ABB RobotStudio station: Lab5_Zhuravlev.rsstn

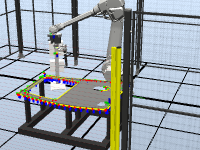
Station GlueStation (saved by RobotStudio 6.8.8307.1040)
Controller IRB4600_20_GlueSystem
  mechanical unit ROB_1: IRB4600_20_250_C_01, 6 joints, base frame (0, 0, 0) mm
Layout (positions relative to the parent item):
  - docking_station [part] at (0, -1345.92, 10) mm, rotated rx 0 ry 0 rz -150 deg
  - SingleDoser [mechanism, from Libraries\SingleDoser.rslib] at (301.98, -1221.72, 1139.56) mm, rotated rx 180 ry -15 rz 15 deg
  - fixture and workpiece [graphiccomponentgroup]
    - door [part]
    - fixture [part]
  - SC_FenceCreator [smart component] at (-1200, -3000, 10) mm
      properties: LengthXside1=4000; LengthXside2=4000; LengthYside1=5300; LengthYside2minus=1500; LengthYside2plus=1500
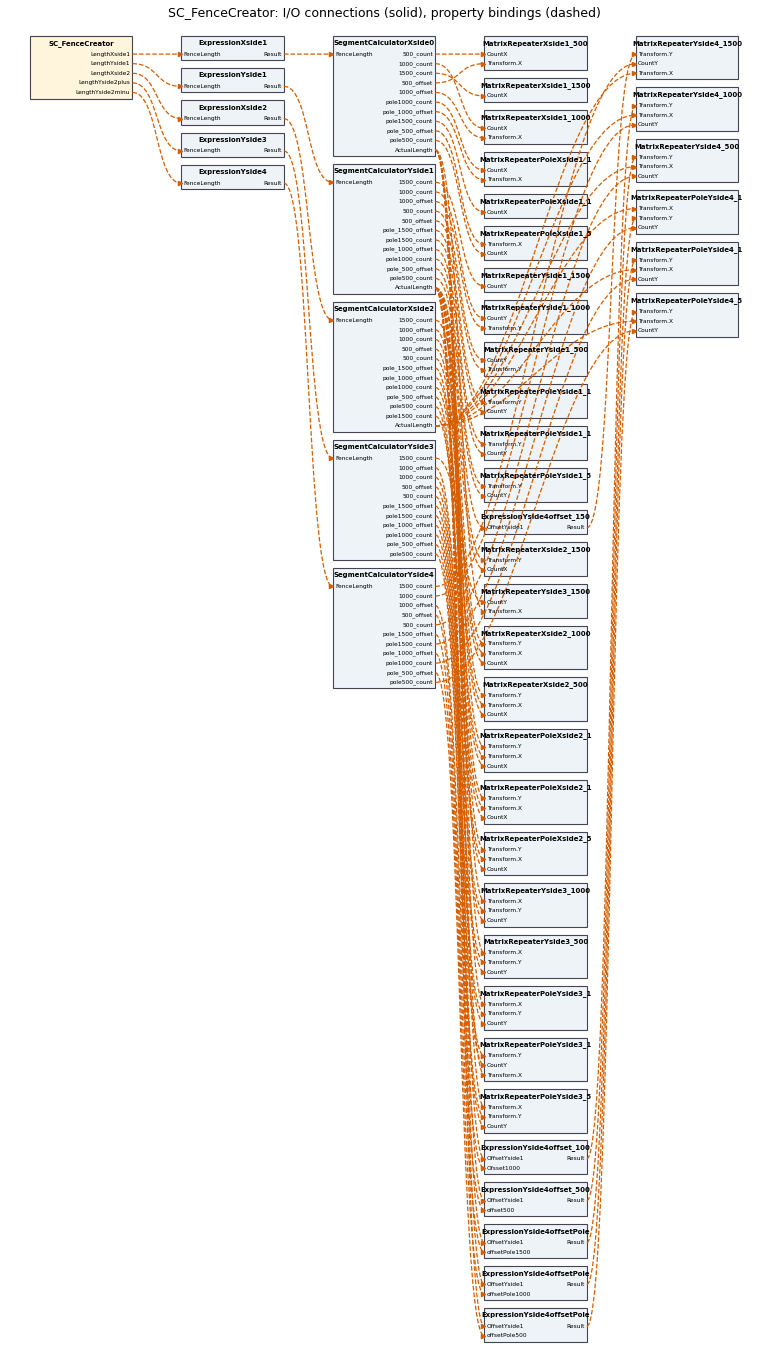
      connections:
        SegmentCalculatorXside0.500_count => MatrixRepeaterXside1_500.CountX
        SegmentCalculatorXside0.1000_count => MatrixRepeaterXside1_1000.CountX
        SegmentCalculatorXside0.1500_count => MatrixRepeaterXside1_1500.CountX
        SegmentCalculatorXside0.500_offset => MatrixRepeaterXside1_500.Transform.X
        SegmentCalculatorXside0.1000_offset => MatrixRepeaterXside1_1000.Transform.X
        SegmentCalculatorXside0.pole1000_count => MatrixRepeaterPoleXside1_1000.CountX
        SegmentCalculatorXside0.pole_1000_offset => MatrixRepeaterPoleXside1_1000.Transform.X
        SegmentCalculatorXside0.pole1500_count => MatrixRepeaterPoleXside1_1500.CountX
        SegmentCalculatorXside0.pole_500_offset => MatrixRepeaterPoleXside1_500.Transform.X
        SegmentCalculatorXside0.pole500_count => MatrixRepeaterPoleXside1_500.CountX
        ExpressionYside1.Result => SegmentCalculatorYside1.FenceLength
        SegmentCalculatorYside1.1500_count => MatrixRepeaterYside1_1500.CountY
        SegmentCalculatorYside1.1000_count => MatrixRepeaterYside1_1000.CountY
        SegmentCalculatorYside1.1000_offset => MatrixRepeaterYside1_1000.Transform.Y
        SegmentCalculatorYside1.500_count => MatrixRepeaterYside1_500.CountY
        SegmentCalculatorYside1.500_offset => MatrixRepeaterYside1_500.Transform.Y
        SegmentCalculatorYside1.pole_1500_offset => MatrixRepeaterPoleYside1_1500.Transform.Y
        SegmentCalculatorYside1.pole1500_count => MatrixRepeaterPoleYside1_1500.CountY
        SegmentCalculatorYside1.pole_1000_offset => MatrixRepeaterPoleYside1_1000.Transform.Y
        SegmentCalculatorYside1.pole1000_count => MatrixRepeaterPoleYside1_1000.CountY
        SegmentCalculatorYside1.pole_500_offset => MatrixRepeaterPoleYside1_500.Transform.Y
        SegmentCalculatorYside1.pole500_count => MatrixRepeaterPoleYside1_500.CountY
        SC_FenceCreator.LengthXside1 => ExpressionXside1.FenceLength
        ExpressionXside2.Result => SegmentCalculatorXside2.FenceLength
        SegmentCalculatorYside1.ActualLength => MatrixRepeaterXside2_1500.Transform.Y
        SegmentCalculatorXside2.1500_count => MatrixRepeaterXside2_1500.CountX
        SegmentCalculatorYside1.ActualLength => MatrixRepeaterXside2_1000.Transform.Y
        SegmentCalculatorXside2.1000_offset => MatrixRepeaterXside2_1000.Transform.X
        SegmentCalculatorXside2.1000_count => MatrixRepeaterXside2_1000.CountX
        SegmentCalculatorYside1.ActualLength => MatrixRepeaterXside2_500.Transform.Y
        SegmentCalculatorXside2.500_offset => MatrixRepeaterXside2_500.Transform.X
        SegmentCalculatorXside2.500_count => MatrixRepeaterXside2_500.CountX
        SegmentCalculatorYside1.ActualLength => MatrixRepeaterPoleXside2_1500.Transform.Y
        SegmentCalculatorXside2.pole_1500_offset => MatrixRepeaterPoleXside2_1500.Transform.X
        SegmentCalculatorYside1.ActualLength => MatrixRepeaterPoleXside2_1000.Transform.Y
        SegmentCalculatorXside2.pole_1000_offset => MatrixRepeaterPoleXside2_1000.Transform.X
        SegmentCalculatorXside2.pole1000_count => MatrixRepeaterPoleXside2_1000.CountX
        SegmentCalculatorYside1.ActualLength => MatrixRepeaterPoleXside2_500.Transform.Y
        SegmentCalculatorXside2.pole_500_offset => MatrixRepeaterPoleXside2_500.Transform.X
        SegmentCalculatorXside2.pole500_count => MatrixRepeaterPoleXside2_500.CountX
        SegmentCalculatorXside2.pole1500_count => MatrixRepeaterPoleXside2_1500.CountX
        SegmentCalculatorYside3.1500_count => MatrixRepeaterYside3_1500.CountY
        ExpressionYside3.Result => SegmentCalculatorYside3.FenceLength
        SegmentCalculatorXside0.ActualLength => MatrixRepeaterYside3_1500.Transform.X
        SegmentCalculatorXside0.ActualLength => MatrixRepeaterYside3_1000.Transform.X
        SegmentCalculatorYside3.1000_offset => MatrixRepeaterYside3_1000.Transform.Y
        SegmentCalculatorYside3.1000_count => MatrixRepeaterYside3_1000.CountY
        SegmentCalculatorXside0.ActualLength => MatrixRepeaterYside3_500.Transform.X
        SegmentCalculatorYside3.500_offset => MatrixRepeaterYside3_500.Transform.Y
        SegmentCalculatorYside3.500_count => MatrixRepeaterYside3_500.CountY
        SegmentCalculatorXside0.ActualLength => MatrixRepeaterPoleYside3_1500.Transform.X
        SegmentCalculatorYside3.pole_1500_offset => MatrixRepeaterPoleYside3_1500.Transform.Y
        SegmentCalculatorYside3.pole1500_count => MatrixRepeaterPoleYside3_1500.CountY
        SegmentCalculatorYside3.pole_1000_offset => MatrixRepeaterPoleYside3_1000.Transform.Y
        SegmentCalculatorYside3.pole1000_count => MatrixRepeaterPoleYside3_1000.CountY
        SegmentCalculatorXside0.ActualLength => MatrixRepeaterPoleYside3_500.Transform.X
        SegmentCalculatorYside3.pole_500_offset => MatrixRepeaterPoleYside3_500.Transform.Y
        SegmentCalculatorYside3.pole500_count => MatrixRepeaterPoleYside3_500.CountY
        SegmentCalculatorXside0.ActualLength => MatrixRepeaterPoleYside3_1000.Transform.X
        ExpressionXside1.Result => SegmentCalculatorXside0.FenceLength
        SC_FenceCreator.LengthYside1 => ExpressionYside1.FenceLength
        SC_FenceCreator.LengthXside2 => ExpressionXside2.FenceLength
        SC_FenceCreator.LengthYside2plus => ExpressionYside3.FenceLength
        SC_FenceCreator.LengthYside2minus => ExpressionYside4.FenceLength
        ExpressionYside4.Result => SegmentCalculatorYside4.FenceLength
        SegmentCalculatorYside1.ActualLength => ExpressionYside4offset_1500.OffsetYside1
        ExpressionYside4offset_1500.Result => MatrixRepeaterYside4_1500.Transform.Y
        SegmentCalculatorYside4.1500_count => MatrixRepeaterYside4_1500.CountY
        SegmentCalculatorXside2.ActualLength => MatrixRepeaterYside4_1500.Transform.X
        SegmentCalculatorYside1.ActualLength => ExpressionYside4offset_1000.OffsetYside1
        ExpressionYside4offset_1000.Result => MatrixRepeaterYside4_1000.Transform.Y
        SegmentCalculatorXside2.ActualLength => MatrixRepeaterYside4_1000.Transform.X
        SegmentCalculatorYside4.1000_count => MatrixRepeaterYside4_1000.CountY
        SegmentCalculatorYside4.1000_offset => ExpressionYside4offset_1000.Ofsset1000
        SegmentCalculatorYside1.ActualLength => ExpressionYside4offset_500.OffsetYside1
        SegmentCalculatorYside4.500_offset => ExpressionYside4offset_500.offset500
        ExpressionYside4offset_500.Result => MatrixRepeaterYside4_500.Transform.Y
        SegmentCalculatorXside2.ActualLength => MatrixRepeaterYside4_500.Transform.X
        SegmentCalculatorYside4.500_count => MatrixRepeaterYside4_500.CountY
        SegmentCalculatorXside2.ActualLength => MatrixRepeaterPoleYside4_1500.Transform.X
        SegmentCalculatorYside1.ActualLength => ExpressionYside4offsetPole_1500.OffsetYside1
        SegmentCalculatorYside4.pole_1500_offset => ExpressionYside4offsetPole_1500.offsetPole1500
        ExpressionYside4offsetPole_1500.Result => MatrixRepeaterPoleYside4_1500.Transform.Y
        SegmentCalculatorYside4.pole1500_count => MatrixRepeaterPoleYside4_1500.CountY
        SegmentCalculatorYside1.ActualLength => ExpressionYside4offsetPole_1000.OffsetYside1
        SegmentCalculatorYside4.pole_1000_offset => ExpressionYside4offsetPole_1000.offsetPole1000
        ExpressionYside4offsetPole_1000.Result => MatrixRepeaterPoleYside4_1000.Transform.Y
        SegmentCalculatorXside2.ActualLength => MatrixRepeaterPoleYside4_1000.Transform.X
        SegmentCalculatorYside4.pole1000_count => MatrixRepeaterPoleYside4_1000.CountY
        SegmentCalculatorYside1.ActualLength => ExpressionYside4offsetPole_500.OffsetYside1
        SegmentCalculatorYside4.pole_500_offset => ExpressionYside4offsetPole_500.offsetPole500
        ExpressionYside4offsetPole_500.Result => MatrixRepeaterPoleYside4_500.Transform.Y
        SegmentCalculatorXside2.ActualLength => MatrixRepeaterPoleYside4_500.Transform.X
        SegmentCalculatorYside4.pole500_count => MatrixRepeaterPoleYside4_500.CountY
    - ExpressionXside1 [smart component, from Libraries\Expression.rslib]
        properties: Expression=FenceLength/1000; FenceLength=4000; Result=4
    - MatrixRepeaterXside1_1500 [smart component, from Libraries\MatrixRepeater.rslib]
        properties: CountX=2; CountY=1; CountZ=1; OffsetX=1.5; OffsetY=0; OffsetZ=0; Source=Panel 2000x1500 X
      - Panel 2000x1500 X [part]
      - Panel 2000x1500 X [part] at (1500, 0, 0) mm
    - MatrixRepeaterXside1_1000 [smart component, from Libraries\MatrixRepeater.rslib] at (3000, 0, 0) mm
        properties: CountX=1; CountY=1; CountZ=1; OffsetX=1; OffsetY=0; OffsetZ=0; Source=Panel 2000x1000 X
      - Panel 2000x1000 X [part]
    - MatrixRepeaterXside1_500 [smart component, from Libraries\MatrixRepeater.rslib] at (4000, 0, 0) mm
        properties: CountX=0; CountY=1; CountZ=1; OffsetX=0.5; OffsetY=0; OffsetZ=0; Source=Panel 2000x500 X
    - MatrixRepeaterPoleXside1_1000 [smart component, from Libraries\MatrixRepeater.rslib] at (4000, 0, 0) mm
        properties: CountX=1; CountY=1; CountZ=1; OffsetX=1; OffsetY=0; OffsetZ=0; Source=Pole
      - Pole [part]
    - Pole [part] at (0, 0, 0) mm
    - SegmentCalculatorXside0 [smart component]
        properties: 1000_count=1; 1000_offset=3; 1500_count=2; 500_count=0; 500_offset=4; ActualLength=4; FenceLength=4; pole_1000_offset=4; pole_1500_offset=0; pole_500_offset=4.5; pole1000_count=1; pole1500_count=3; pole500_count=0; SideNo=0
    - MatrixRepeaterPoleXside1_1500 [smart component, from Libraries\MatrixRepeater.rslib]
        properties: CountX=3; CountY=1; CountZ=1; OffsetX=1.5; OffsetY=0; OffsetZ=1; Source=Pole
      - Pole [part]
      - Pole [part] at (1500, 0, 0) mm
      - Pole [part] at (3000, 0, 0) mm
    - MatrixRepeaterPoleXside1_500 [smart component, from Libraries\MatrixRepeater.rslib] at (4500, 0, 0) mm
        properties: CountX=0; CountY=1; CountZ=1; OffsetX=0.5; OffsetY=0; OffsetZ=0; Source=Pole
    - ExpressionYside1 [smart component, from Libraries\Expression.rslib]
        properties: Expression=FenceLength/1000; FenceLength=5300; Result=5.3
    - MatrixRepeaterYside1_1500 [smart component, from Libraries\MatrixRepeater.rslib]
        properties: CountX=1; CountY=3; CountZ=1; OffsetX=0; OffsetY=1.5; OffsetZ=0; Source=Panel 2000x1500 Y
      - Panel 2000x1500 Y [part]
      - Panel 2000x1500 Y [part] at (0, 1500, 0) mm
      - Panel 2000x1500 Y [part] at (0, 3000, 0) mm
    - MatrixRepeaterYside1_1000 [smart component, from Libraries\MatrixRepeater.rslib] at (0, 4500, 0) mm
        properties: CountX=1; CountY=1; CountZ=1; OffsetX=0; OffsetY=1; OffsetZ=0; Source=Panel 2000x1000 Y
      - Panel 2000x1000 Y [part]
    - MatrixRepeaterYside1_500 [smart component, from Libraries\MatrixRepeater.rslib] at (0, 5500, 0) mm
        properties: CountX=1; CountY=0; CountZ=1; OffsetX=0; OffsetY=0.5; OffsetZ=0; Source=Panel 2000x500 Y
    - PoleYside1 [part] at (0, 0, 0) mm
    - MatrixRepeaterPoleYside1_1500 [smart component, from Libraries\MatrixRepeater.rslib] at (0, 1500, 0) mm
        properties: CountX=1; CountY=3; CountZ=1; OffsetX=0; OffsetY=1.5; OffsetZ=0; Source=PoleYside1
      - PoleYside1 [part]
      - PoleYside1 [part] at (0, 1500, 0) mm
      - PoleYside1 [part] at (0, 3000, 0) mm
    - SegmentCalculatorYside1 [smart component]
        properties: 1000_count=1; 1000_offset=4.5; 1500_count=3; 500_count=0; 500_offset=5.5; ActualLength=5.5; FenceLength=5.3; pole_1000_offset=5.5; pole_1500_offset=1.5; pole_500_offset=6; pole1000_count=1; pole1500_count=3; pole500_count=0; SideNo=1
    - MatrixRepeaterPoleYside1_1000 [smart component, from Libraries\MatrixRepeater.rslib] at (0, 5500, 0) mm
        properties: CountX=1; CountY=1; CountZ=1; OffsetX=0; OffsetY=1; OffsetZ=0; Source=PoleYside1
      - PoleYside1 [part]
    - MatrixRepeaterPoleYside1_500 [smart component, from Libraries\MatrixRepeater.rslib] at (0, 6000, 0) mm
        properties: CountX=1; CountY=0; CountZ=1; OffsetX=0; OffsetY=0.5; OffsetZ=0; Source=PoleYside1
    - PoleXside2 [part] at (0, 0, 0) mm
    - PoleYside3 [part] at (0, 0, 0) mm
    - ExpressionXside2 [smart component, from Libraries\Expression.rslib]
        properties: Expression=FenceLength/1000; FenceLength=4000; Result=4
    - SegmentCalculatorXside2 [smart component]
        properties: 1000_count=1; 1000_offset=3; 1500_count=2; 500_count=0; 500_offset=4; ActualLength=4; FenceLength=4; pole_1000_offset=4; pole_1500_offset=1.5; pole_500_offset=4.5; pole1000_count=1; pole1500_count=2; pole500_count=0; SideNo=2
    - MatrixRepeaterXside2_1500 [smart component, from Libraries\MatrixRepeater.rslib] at (0, 5500, 0) mm
        properties: CountX=2; CountY=1; CountZ=1; OffsetX=1.5; OffsetY=0; OffsetZ=0; Source=Panel 2000x1500 X
      - Panel 2000x1500 X [part]
      - Panel 2000x1500 X [part] at (1500, 0, 0) mm
    - MatrixRepeaterXside2_1000 [smart component, from Libraries\MatrixRepeater.rslib] at (3000, 5500, 0) mm
        properties: CountX=1; CountY=1; CountZ=1; OffsetX=1; OffsetY=0; OffsetZ=0; Source=Panel 2000x1000 X
      - Panel 2000x1000 X [part]
    - MatrixRepeaterXside2_500 [smart component, from Libraries\MatrixRepeater.rslib] at (4000, 5500, 0) mm
        properties: CountX=0; CountY=1; CountZ=1; OffsetX=0.5; OffsetY=0; OffsetZ=0; Source=Panel 2000x500 X
    - MatrixRepeaterPoleXside2_1500 [smart component, from Libraries\MatrixRepeater.rslib] at (1500, 5500, 0) mm
        properties: CountX=2; CountY=1; CountZ=1; OffsetX=1.5; OffsetY=0; OffsetZ=0; Source=PoleXside2
      - PoleXside2 [part]
      - PoleXside2 [part] at (1500, 0, 0) mm
    - MatrixRepeaterPoleXside2_1000 [smart component, from Libraries\MatrixRepeater.rslib] at (4000, 5500, 0) mm
        properties: CountX=1; CountY=1; CountZ=1; OffsetX=1; OffsetY=0; OffsetZ=0; Source=PoleXside2
      - PoleXside2 [part]
    - MatrixRepeaterPoleXside2_500 [smart component, from Libraries\MatrixRepeater.rslib] at (4500, 5500, 0) mm
        properties: CountX=0; CountY=1; CountZ=1; OffsetX=0.5; OffsetY=0; OffsetZ=0; Source=PoleXside2
    - SegmentCalculatorYside3 [smart component]
        properties: 1000_count=0; 1000_offset=1.5; 1500_count=1; 500_count=0; 500_offset=1.5; ActualLength=1.5; FenceLength=1.5; pole_1000_offset=2.5; pole_1500_offset=1.5; pole_500_offset=2; pole1000_count=0; pole1500_count=1; pole500_count=0; SideNo=3
    - ExpressionYside3 [smart component]
        properties: Expression=FenceLength/1000; FenceLength=1500; Result=1.5
    - MatrixRepeaterYside3_1500 [smart component] at (4000, 0, 0) mm
        properties: CountX=1; CountY=1; CountZ=1; OffsetX=0; OffsetY=1.5; OffsetZ=0; Source=Panel 2000x1500 Y
      - Panel 2000x1500 Y [part]
    - MatrixRepeaterYside3_1000 [smart component] at (4000, 1500, 0) mm
        properties: CountX=1; CountY=0; CountZ=1; OffsetX=0; OffsetY=1; OffsetZ=0; Source=Panel 2000x1000 Y
    - MatrixRepeaterYside3_500 [smart component] at (4000, 1500, 0) mm
        properties: CountX=1; CountY=0; CountZ=1; OffsetX=0; OffsetY=0.5; OffsetZ=0; Source=Panel 2000x500 Y
    - MatrixRepeaterPoleYside3_1500 [smart component] at (4000, 1500, 0) mm
        properties: CountX=1; CountY=1; CountZ=1; OffsetX=0; OffsetY=1.5; OffsetZ=0; Source=PoleYside3
      - PoleYside3 [part]
    - MatrixRepeaterPoleYside3_1000 [smart component] at (4000, 2500, 0) mm
        properties: CountX=1; CountY=0; CountZ=1; OffsetX=0; OffsetY=1; OffsetZ=0; Source=PoleYside3
    - MatrixRepeaterPoleYside3_500 [smart component] at (4000, 2000, 0) mm
        properties: CountX=1; CountY=0; CountZ=1; OffsetX=0; OffsetY=0.5; OffsetZ=0; Source=PoleYside3
    - ExpressionYside4 [smart component, from Libraries\Expression.rslib]
        properties: Expression=FenceLength/1000; FenceLength=1500; Result=1.5
    - SegmentCalculatorYside4 [smart component]
        properties: 1000_count=0; 1000_offset=1.5; 1500_count=1; 500_count=0; 500_offset=1.5; ActualLength=1.5; FenceLength=1.5; pole_1000_offset=2.5; pole_1500_offset=1.5; pole_500_offset=2; pole1000_count=0; pole1500_count=1; pole500_count=0; SideNo=4
    - MatrixRepeaterYside4_1500 [smart component, from Libraries\MatrixRepeater.rslib] at (4000, 4000, 0) mm
        properties: CountX=1; CountY=1; CountZ=1; OffsetX=0; OffsetY=-1.5; OffsetZ=0; Source=Panel 2000x1500 Y
      - Panel 2000x1500 Y [part]
    - ExpressionYside4offset_1500 [smart component, from Libraries\Expression.rslib]
        properties: Expression=OffsetYside1-1.5; OffsetYside1=5.5; Result=4
    - ExpressionYside4offset_1000 [smart component, from Libraries\Expression.rslib]
        properties: Expression=OffsetYside1-Ofsset1000-1; OffsetYside1=5.5; Ofsset1000=1.5; Result=3
    - MatrixRepeaterYside4_1000 [smart component, from Libraries\MatrixRepeater.rslib] at (4000, 3000, 0) mm
        properties: CountX=1; CountY=0; CountZ=1; OffsetX=0; OffsetY=-1; OffsetZ=0; Source=Panel 2000x1000 Y
    - ExpressionYside4offset_500 [smart component, from Libraries\Expression.rslib]
        properties: Expression=OffsetYside1-offset500-0.5; offset500=1.5; OffsetYside1=5.5; Result=3.5
    - MatrixRepeaterYside4_500 [smart component, from Libraries\MatrixRepeater.rslib] at (4000, 3500, 0) mm
        properties: CountX=1; CountY=0; CountZ=1; OffsetX=0; OffsetY=-0.5; OffsetZ=0; Source=Panel 2000x500 Y
    - MatrixRepeaterPoleYside4_1500 [smart component, from Libraries\MatrixRepeater.rslib] at (4000, 4000, 0) mm
        properties: CountX=1; CountY=1; CountZ=1; OffsetX=0; OffsetY=-1.5; OffsetZ=0; Source=PoleYside3
      - PoleYside3 [part]
    - ExpressionYside4offsetPole_1500 [smart component, from Libraries\Expression.rslib]
        properties: Expression=OffsetYside1-offsetPole1500; offsetPole1500=1.5; OffsetYside1=5.5; Result=4
    - ExpressionYside4offsetPole_1000 [smart component, from Libraries\Expression.rslib]
        properties: Expression=OffsetYside1-offsetPole1000; offsetPole1000=2.5; OffsetYside1=5.5; Result=3
    - MatrixRepeaterPoleYside4_1000 [smart component, from Libraries\MatrixRepeater.rslib] at (4000, 3000, 0) mm
        properties: CountX=1; CountY=0; CountZ=1; OffsetX=0; OffsetY=-1; OffsetZ=0; Source=PoleYside3
    - ExpressionYside4offsetPole_500 [smart component, from Libraries\Expression.rslib]
        properties: Expression=OffsetYside1-offsetPole500; offsetPole500=2; OffsetYside1=5.5; Result=3.5
    - MatrixRepeaterPoleYside4_500 [smart component, from Libraries\MatrixRepeater.rslib] at (4000, 3500, 0) mm
        properties: CountX=1; CountY=0; CountZ=1; OffsetX=0; OffsetY=-0.5; OffsetZ=0; Source=PoleYside3
    - Panel 2000x1000 X [part]
    - Panel 2000x1500 X [part]
    - Panel 2000x500 X [part]
    - Panel 2000x1000 Y [part]
    - Panel 2000x1500 Y [part]
    - Panel 2000x500 Y [part]
  - SC_LightGuard [smart component] at (2800, -1416, 10) mm, rotated rx 0 ry 0 rz 90 deg
      properties: GuardDistance=2330; vecPosition=[0 0 0]; vecOrientation=[0 0 0]
      signals: DI UpdateDistance, DI diGuardOn
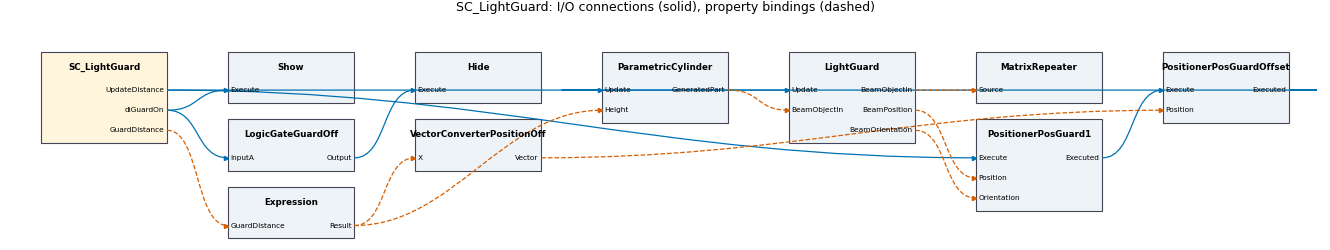
      connections:
        SC_LightGuard.UpdateDistance -> LightGuard.Update
        SC_LightGuard.UpdateDistance -> PositionerPosGuard1.Execute
        PositionerPosGuard1.Executed -> PositionerPosGuardOffset.Execute
        PositionerPosGuardOffset.Executed -> ParametricCylinder.Update
        SC_LightGuard.diGuardOn -> Show.Execute
        SC_LightGuard.diGuardOn -> LogicGateGuardOff.InputA
        LogicGateGuardOff.Output -> Hide.Execute
        SC_LightGuard.GuardDistance => Expression.GuardDistance
        Expression.Result => VectorConverterPositionOffset.X
        VectorConverterPositionOffset.Vector => PositionerPosGuardOffset.Position
        Expression.Result => ParametricCylinder.Height
        ParametricCylinder.GeneratedPart => LightGuard.BeamObjectIn
        LightGuard.BeamObjectIn => MatrixRepeater.Source
        LightGuard.BeamPosition => PositionerPosGuard1.Position
        LightGuard.BeamOrientation => PositionerPosGuard1.Orientation
    - light_guard2 [part] at (2330, 0, 0) mm
    - light_guard1 [part]
    - PositionerPosGuard1 [smart component]
        properties: Object=light_guard2; Position=[2.8 -1.416 0.01]; Orientation=[0 0 1.5707963267949]; Reference=Global; ReferenceObject=SC_LightGuard
        signals: DI Execute, DO Executed
    - Expression [smart component]
        properties: Expression=GuardDistance/1000; Result=2.33; GuardDistance=2330
    - PositionerPosGuardOffset [smart component]
        properties: Object=light_guard2; Position=[2.33 0 0]; Orientation=[0 0 0]; Reference=Local; ReferenceObject=(none)
        signals: DI Execute, DO Executed
    - VectorConverterPositionOffset [smart component]
        properties: X=2.33; Y=0; Z=0; Vector=[2.33 0 0]
    - ParametricCylinder [smart component] at (0, 0, 200) mm, rotated rx 0 ry 90 rz 0 deg
        properties: Radius=0.002; Height=2.33; GeneratedPart=GeneratedPart; KeepGeometry=true
        signals: DI Update
      - GeneratedPart [part]
    - MatrixRepeater [smart component] at (0, 0, 200) mm, rotated rx 0 ry 90 rz 0 deg
        properties: Source=GeneratedPart; CountX=32; CountY=1; CountZ=1; OffsetX=-0.05; OffsetY=0; OffsetZ=0
      - GeneratedPart [part]
      - GeneratedPart [part] at (-50, 0, 0) mm
      - GeneratedPart [part] at (-100, 0, 0) mm
      - GeneratedPart [part] at (-150, 0, 0) mm
      - GeneratedPart [part] at (-200, 0, 0) mm
      - GeneratedPart [part] at (-250, 0, 0) mm
      - GeneratedPart [part] at (-300, 0, 0) mm
      - GeneratedPart [part] at (-350, 0, 0) mm
      - GeneratedPart [part] at (-400, 0, 0) mm
      - GeneratedPart [part] at (-450, 0, 0) mm
      - GeneratedPart [part] at (-500, 0, 0) mm
      - GeneratedPart [part] at (-550, 0, 0) mm
      - GeneratedPart [part] at (-600, 0, 0) mm
      - GeneratedPart [part] at (-650, 0, 0) mm
      - GeneratedPart [part] at (-700, 0, 0) mm
      - GeneratedPart [part] at (-750, 0, 0) mm
      - GeneratedPart [part] at (-800, 0, 0) mm
      - GeneratedPart [part] at (-850, 0, 0) mm
      - GeneratedPart [part] at (-900, 0, 0) mm
      - GeneratedPart [part] at (-950, 0, 0) mm
      - GeneratedPart [part] at (-1000, 0, 0) mm
      - GeneratedPart [part] at (-1050, 0, 0) mm
      - GeneratedPart [part] at (-1100, 0, 0) mm
      - GeneratedPart [part] at (-1150, 0, 0) mm
      - GeneratedPart [part] at (-1200, 0, 0) mm
      - GeneratedPart [part] at (-1250, 0, 0) mm
      - GeneratedPart [part] at (-1300, 0, 0) mm
      - GeneratedPart [part] at (-1350, 0, 0) mm
      - GeneratedPart [part] at (-1400, 0, 0) mm
      - GeneratedPart [part] at (-1450, 0, 0) mm
      - GeneratedPart [part] at (-1500, 0, 0) mm
      - GeneratedPart [part] at (-1550, 0, 0) mm
    - Show [smart component]
        properties: Object=MatrixRepeater
        signals: DI Execute, DO Executed
    - Hide [smart component]
        properties: Object=MatrixRepeater
        signals: DI Execute, DO Executed
    - LogicGateGuardOff [smart component]
        properties: Operator=NOT; Delay=0
        signals: DI InputA, DI InputB, DO Output
    - LightGuard [smart component]
        properties: BeamObjectIn=GeneratedPart; LightGuard=light_guard1; BeamObjectOut=GeneratedPart; BeamPosition=[2.8 -1.416 0.01]; BeamOrientation=[0 0 1.5707963267949]
        signals: DI Update
  - IRB4600_20_250_C_01 [mechanism, from Robots\IRB4600_20_250_C_G_01.rslib] at (0, 0, 0) mm; joint values [-1.3459, -0.0956, 0.5335, 0.2862, 1.1582, 1.4151] (rad or m)
  - Part_1 [part] at (1465.26, 1021.34, 716.54) mm, rotated rx 93.78 ry 0.08 rz 0 deg
  - Part_2 [part] at (1465.26, 1021.34, 716.54) mm, rotated rx 93.78 ry 0.08 rz 0 deg
Attachment: SingleDoser is attached to IRB4600_20_250_C_01 / Link6
Collision set CollisionSet_1: SingleDoser against fixture and workpiece, near miss 0.004 m
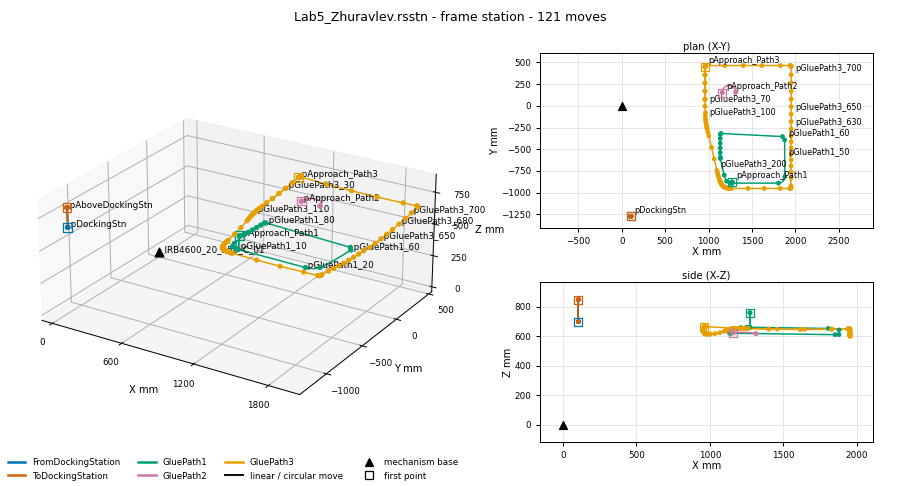
[picture p0: tool path of Lab5_Zhuravlev.rsstn in frame station, 121 of 121 moves have a stored position in this frame; points joined in program order, loops and branches not executed]
Targets, tools, work objects and paths stored in the station, written as RAPID:
! task T_ROB1
MODULE modRobotStudio
  CONST robtarget pDockingStn:=[[-6.21722435,13.985562095,-127.5],[0,0.737075919,0.675809951,0],[-1,0,0,0],[9E+09,9E+09,9E+09,9E+09,9E+09,9E+09]];
  CONST robtarget pAboveDockingStn:=[[-6.217297914,13.985583992,22.500016978],[-0.000000026,0.737075879,0.675809995,-0.000000022],[-1,0,0,0],[9E+09,9E+09,9E+09,9E+09,9E+09,9E+09]];
  PROC FromDockingStation()
    MoveJ pDockingStn,v200,z1,tNozzle\WObj:=wobjDockingStn;
    MoveL pAboveDockingStn,v200,z1,tNozzle\WObj:=wobjDockingStn;
  ENDPROC
  PROC ToDockingStation()
    MoveL pAboveDockingStn,v1000,z1,tNozzle\WObj:=wobjDockingStn;
    MoveL pDockingStn,v200,fine,tNozzle\WObj:=wobjDockingStn;
  ENDPROC
  PROC GluePath1()
    MoveL pApproach_Path1,v1000,z100,tNozzle\WObj:=WobjFixture;
    MoveL pGluePath1_10,v300,z1,tNozzle\WObj:=WobjFixture;
    MoveL pGluePath1_20,v300,z1,tNozzle\WObj:=WobjFixture;
    MoveC pGluePath1_30,pGluePath1_40,v300,z1,tNozzle\WObj:=WobjFixture;
    MoveC pGluePath1_50,pGluePath1_60,v300,z1,tNozzle\WObj:=WobjFixture;
    MoveL pGluePath1_70,v300,z1,tNozzle\WObj:=WobjFixture;
    MoveL pGluePath1_80,v300,z1,tNozzle\WObj:=WobjFixture;
    MoveC pGluePath1_90,pGluePath1_100,v300,z1,tNozzle\WObj:=WobjFixture;
    MoveL pGluePath1_110,v300,z1,tNozzle\WObj:=WobjFixture;
    MoveL pGluePath1_120,v300,z1,tNozzle\WObj:=WobjFixture;
    MoveL pGluePath1_130,v300,z1,tNozzle\WObj:=WobjFixture;
    MoveL pGluePath1_140,v300,z1,tNozzle\WObj:=WobjFixture;
    MoveL pGluePath1_150,v300,z1,tNozzle\WObj:=WobjFixture;
    MoveL pGluePath1_160,v300,z1,tNozzle\WObj:=WobjFixture;
    MoveL pGluePath1_170,v300,z1,tNozzle\WObj:=WobjFixture;
    MoveC pGluePath1_180,pGluePath1_190,v300,z1,tNozzle\WObj:=WobjFixture;
    MoveC pGluePath1_200,pGluePath1_210,v300,z1,tNozzle\WObj:=WobjFixture;
    MoveC pGluePath1_220,pGluePath1_230,v300,z1,tNozzle\WObj:=WobjFixture;
    MoveL pGluePath1_240,v300,z1,tNozzle\WObj:=WobjFixture;
    MoveL pGluePath1_250,v300,z1,tNozzle\WObj:=WobjFixture;
    MoveL pDepart_Path1,v1000,z100,tNozzle\WObj:=WobjFixture;
  ENDPROC
  PROC GluePath2()
    MoveL pApproach_Path2,v1000,z100,tNozzle\WObj:=WobjFixture;
    MoveL pGluePath2_10,v300,z1,tNozzle\WObj:=WobjFixture;
    MoveC pGluePath2_20,pGluePath2_30,v300,z1,tNozzle\WObj:=WobjFixture;
    MoveL pDepart_Path2,v1000,z100,tNozzle\WObj:=WobjFixture;
  ENDPROC
  PROC GluePath3()
    MoveL pApproach_Path3,v1000,z100,tNozzle\WObj:=WobjFixture;
    MoveL pGluePath3_10,v300,z1,tNozzle\WObj:=WobjFixture;
    MoveL pGluePath3_20,v300,z1,tNozzle\WObj:=WobjFixture;
    MoveL pGluePath3_30,v300,z1,tNozzle\WObj:=WobjFixture;
    MoveL pGluePath3_40,v300,z1,tNozzle\WObj:=WobjFixture;
    MoveL pGluePath3_50,v300,z1,tNozzle\WObj:=WobjFixture;
    MoveL pGluePath3_70,v300,z1,tNozzle\WObj:=WobjFixture;
    MoveL pGluePath3_80,v300,z1,tNozzle\WObj:=WobjFixture;
    MoveL pGluePath3_90,v300,z1,tNozzle\WObj:=WobjFixture;
    MoveL pGluePath3_100,v300,z1,tNozzle\WObj:=WobjFixture;
    MoveL pGluePath3_110,v300,z1,tNozzle\WObj:=WobjFixture;
    MoveL pGluePath3_120,v300,z1,tNozzle\WObj:=WobjFixture;
    MoveL pGluePath3_130,v300,z1,tNozzle\WObj:=WobjFixture;
    MoveL pGluePath3_140,v300,z1,tNozzle\WObj:=WobjFixture;
    MoveL pGluePath3_150,v300,z1,tNozzle\WObj:=WobjFixture;
    MoveL pGluePath3_160,v300,z1,tNozzle\WObj:=WobjFixture;
    MoveL pGluePath3_170,v300,z1,tNozzle\WObj:=WobjFixture;
    MoveL pGluePath3_180,v300,z1,tNozzle\WObj:=WobjFixture;
    MoveL pGluePath3_190,v300,z1,tNozzle\WObj:=WobjFixture;
    MoveL pGluePath3_200,v300,z1,tNozzle\WObj:=WobjFixture;
    MoveL pGluePath3_210,v300,z1,tNozzle\WObj:=WobjFixture;
    MoveL pGluePath3_220,v300,z1,tNozzle\WObj:=WobjFixture;
    MoveL pGluePath3_230,v300,z1,tNozzle\WObj:=WobjFixture;
    MoveL pGluePath3_240,v300,z1,tNozzle\WObj:=WobjFixture;
    MoveL pGluePath3_250,v300,z1,tNozzle\WObj:=WobjFixture;
    MoveL pGluePath3_260,v300,z1,tNozzle\WObj:=WobjFixture;
    MoveL pGluePath3_270,v300,z1,tNozzle\WObj:=WobjFixture;
    MoveL pGluePath3_280,v300,z1,tNozzle\WObj:=WobjFixture;
    MoveL pGluePath3_290,v300,z1,tNozzle\WObj:=WobjFixture;
    MoveL pGluePath3_300,v300,z1,tNozzle\WObj:=WobjFixture;
    MoveL pGluePath3_310,v300,z1,tNozzle\WObj:=WobjFixture;
    MoveL pGluePath3_320,v300,z1,tNozzle\WObj:=WobjFixture;
    MoveL pGluePath3_330,v300,z1,tNozzle\WObj:=WobjFixture;
    MoveL pGluePath3_340,v300,z1,tNozzle\WObj:=WobjFixture;
    MoveL pGluePath3_350,v300,z1,tNozzle\WObj:=WobjFixture;
    MoveL pGluePath3_360,v300,z1,tNozzle\WObj:=WobjFixture;
    MoveL pGluePath3_370,v300,z1,tNozzle\WObj:=WobjFixture;
    MoveL pGluePath3_380,v300,z1,tNozzle\WObj:=WobjFixture;
    MoveL pGluePath3_390,v300,z1,tNozzle\WObj:=WobjFixture;
    MoveL pGluePath3_400,v300,z1,tNozzle\WObj:=WobjFixture;
    MoveL pGluePath3_410,v300,z1,tNozzle\WObj:=WobjFixture;
    MoveL pGluePath3_420,v300,z1,tNozzle\WObj:=WobjFixture;
    MoveL pGluePath3_430,v300,z1,tNozzle\WObj:=WobjFixture;
    MoveL pGluePath3_440,v300,z1,tNozzle\WObj:=WobjFixture;
    MoveL pGluePath3_450,v300,z1,tNozzle\WObj:=WobjFixture;
    MoveL pGluePath3_460,v300,z1,tNozzle\WObj:=WobjFixture;
    MoveL pGluePath3_470,v300,z1,tNozzle\WObj:=WobjFixture;
    MoveL pGluePath3_480,v300,z1,tNozzle\WObj:=WobjFixture;
    MoveL pGluePath3_490,v300,z1,tNozzle\WObj:=WobjFixture;
    MoveL pGluePath3_500,v300,z1,tNozzle\WObj:=WobjFixture;
    MoveL pGluePath3_510,v300,z1,tNozzle\WObj:=WobjFixture;
    MoveL pGluePath3_520,v300,z1,tNozzle\WObj:=WobjFixture;
    MoveL pGluePath3_530,v300,z1,tNozzle\WObj:=WobjFixture;
    MoveL pGluePath3_550,v300,z1,tNozzle\WObj:=WobjFixture;
    MoveL pGluePath3_560,v300,z1,tNozzle\WObj:=WobjFixture;
    MoveL pGluePath3_570,v300,z1,tNozzle\WObj:=WobjFixture;
    MoveL pGluePath3_580,v300,z1,tNozzle\WObj:=WobjFixture;
    MoveL pGluePath3_590,v300,z1,tNozzle\WObj:=WobjFixture;
    MoveL pGluePath3_600,v300,z1,tNozzle\WObj:=WobjFixture;
    MoveL pGluePath3_610,v300,z1,tNozzle\WObj:=WobjFixture;
    MoveL pGluePath3_620,v300,z1,tNozzle\WObj:=WobjFixture;
    MoveL pGluePath3_630,v300,z1,tNozzle\WObj:=WobjFixture;
    MoveL pGluePath3_640,v300,z1,tNozzle\WObj:=WobjFixture;
    MoveL pGluePath3_650,v300,z1,tNozzle\WObj:=WobjFixture;
    MoveL pGluePath3_660,v300,z1,tNozzle\WObj:=WobjFixture;
    MoveL pGluePath3_670,v300,z1,tNozzle\WObj:=WobjFixture;
    MoveL pGluePath3_680,v300,z1,tNozzle\WObj:=WobjFixture;
    MoveL pGluePath3_690,v300,z1,tNozzle\WObj:=WobjFixture;
    MoveL pGluePath3_700,v300,z1,tNozzle\WObj:=WobjFixture;
    MoveL pGluePath3_710,v300,z1,tNozzle\WObj:=WobjFixture;
    MoveL pGluePath3_720,v300,z1,tNozzle\WObj:=WobjFixture;
    MoveL pGluePath3_730,v300,z1,tNozzle\WObj:=WobjFixture;
    MoveL pGluePath3_740,v300,z1,tNozzle\WObj:=WobjFixture;
    MoveL pGluePath3_750,v300,z1,tNozzle\WObj:=WobjFixture;
    MoveL pGluePath3_760,v300,z1,tNozzle\WObj:=WobjFixture;
    MoveL pGluePath3_770,v300,z1,tNozzle\WObj:=WobjFixture;
    MoveL pGluePath3_780,v300,z1,tNozzle\WObj:=WobjFixture;
    MoveL pGluePath3_790,v300,z1,tNozzle\WObj:=WobjFixture;
    MoveL pGluePath3_800,v300,z1,tNozzle\WObj:=WobjFixture;
    MoveL pGluePath3_810,v300,z1,tNozzle\WObj:=WobjFixture;
    MoveL pGluePath3_820,v300,z1,tNozzle\WObj:=WobjFixture;
    MoveL pGluePath3_830,v300,z1,tNozzle\WObj:=WobjFixture;
    MoveL pGluePath3_840,v300,z1,tNozzle\WObj:=WobjFixture;
    MoveL pGluePath3_850,v300,z1,tNozzle\WObj:=WobjFixture;
    MoveL pGluePath3_860,v300,z1,tNozzle\WObj:=WobjFixture;
    MoveL pGluePath3_870,v300,z1,tNozzle\WObj:=WobjFixture;
    MoveL pGluePath3_880,v300,z1,tNozzle\WObj:=WobjFixture;
    MoveL pDepart_Path3,v1000,z100,tNozzle\WObj:=WobjFixture;
  ENDPROC
  PROC main()
    FromDockingStation;
    GluePath1;
    GluePath2;
    GluePath3;
    ToDockingStation;
  ENDPROC
ENDMODULE

! task T_ROB1
MODULE modCalibData
  TASK PERS wobjdata wobjDockingStn:=[FALSE,TRUE,"",[[93.58826629,-1285.222736121,827.125],[0.818981032,0,0,-0.57382059]],[[0,0,0],[1,0,0,0]]];
  PERS tooldata tNozzle:=[TRUE,[[-311.236392018,0,372.060957775],[0.991444861,0,-0.130526192,0]],[10,[-216.957886762,-4.684934403,103.554004337],[1,0,0,0],0,0,0]];
  TASK PERS wobjdata WobjFixture:=[FALSE,TRUE,"",[[0,0,0],[1,0,0,0]],[[1777.777536733,440.116087079,662.27738287],[0.001576647,-0.002969945,-0.000677106,-0.999994118]]];
ENDMODULE

! task T_ROB1
MODULE Module1
  CONST robtarget pGluePath1_10:=[[510.889716888,1330.321452608,-5.755706549],[0.004277461,0.000888769,0.997748318,0.066926884],[-1,0,1,0],[9E+09,9E+09,9E+09,9E+09,9E+09,9E+09]];
  CONST robtarget pGluePath1_20:=[[-24.026746697,1331.547210356,-10.262043177],[0.004277457,0.000888764,0.997748249,0.066927907],[-1,-1,1,0],[9E+09,9E+09,9E+09,9E+09,9E+09,9E+09]];
  CONST robtarget pGluePath1_30:=[[-75.819066703,1310.049473712,-13.577364347],[0.00427561,0.000898378,0.997896025,0.064687214],[-1,-1,1,0],[9E+09,9E+09,9E+09,9E+09,9E+09,9E+09]];
  CONST robtarget pGluePath1_40:=[[-97.063186424,1258.474377763,-20.210946508],[0.004271118,0.000921316,0.998228583,0.05933468],[-1,-1,1,0],[9E+09,9E+09,9E+09,9E+09,9E+09,9E+09]];
  CONST robtarget pGluePath1_50:=[[-97.374706717,1045.953440443,-40.56745714],[0.004250242,0.00102039,0.999338131,0.036113626],[-1,-1,1,0],[9E+09,9E+09,9E+09,9E+09,9E+09,9E+09]];
  CONST robtarget pGluePath1_60:=[[-97.771486488,832.718195899,-51.025208345],[0.004227066,0.00111885,0.999907627,0.012869259],[-1,0,1,0],[9E+09,9E+09,9E+09,9E+09,9E+09,9E+09]];
  CONST robtarget pGluePath1_70:=[[-72.219006167,794.539727769,-51.633047149],[0.00422295,0.001135325,0.999950266,0.008963479],[-1,0,1,0],[9E+09,9E+09,9E+09,9E+09,9E+09,9E+09]];
  CONST robtarget pGluePath1_80:=[[635.452858017,756.9477876,-46.156535376],[0.004218982,0.001151063,0.999976773,0.005227693],[-1,0,1,0],[9E+09,9E+09,9E+09,9E+09,9E+09,9E+09]];
  CONST robtarget pGluePath1_90:=[[642.120480193,759.42233876,-46.075003727],[0.004219144,0.001150428,0.999975972,0.005378644],[-1,0,1,0],[9E+09,9E+09,9E+09,9E+09,9E+09,9E+09]];
  CONST robtarget pGluePath1_100:=[[644.923000067,765.954849253,-45.979653791],[0.004219569,0.001148758,0.999973762,0.00577507],[-1,0,1,0],[9E+09,9E+09,9E+09,9E+09,9E+09,9E+09]];
  CONST robtarget pGluePath1_110:=[[645.024650126,813.620213836,-45.180818125],[0.004225091,0.001126856,0.999930246,0.010971856],[-1,0,1,0],[9E+09,9E+09,9E+09,9E+09,9E+09,9E+09]];
  CONST robtarget pGluePath1_120:=[[645.136472361,868.489649078,-43.64770765],[0.004231307,0.001101608,0.999846746,0.016951874],[-1,0,1,0],[9E+09,9E+09,9E+09,9E+09,9E+09,9E+09]];
  CONST robtarget pGluePath1_130:=[[645.242715228,923.336821184,-41.458561752],[0.004237373,0.001076326,0.999727534,0.022929091],[-1,0,1,0],[9E+09,9E+09,9E+09,9E+09,9E+09,9E+09]];
  CONST robtarget pGluePath1_140:=[[645.343365182,978.153898711,-38.613887486],[0.00424329,0.001051005,0.999572629,0.02890415],[-1,0,1,0],[9E+09,9E+09,9E+09,9E+09,9E+09,9E+09]];
  CONST robtarget pGluePath1_150:=[[645.438408681,1032.933050284,-35.114191912],[0.004249058,0.001025643,0.999382029,0.034877692],[-1,0,1,0],[9E+09,9E+09,9E+09,9E+09,9E+09,9E+09]];
  CONST robtarget pGluePath1_160:=[[645.124582284,1038.956086956,-34.692049047],[0.00424964,0.001023049,0.999360541,0.035488076],[-1,0,1,0],[9E+09,9E+09,9E+09,9E+09,9E+09,9E+09]];
  CONST robtarget pGluePath1_170:=[[644.1683715,1044.911297822,-34.27245051],[0.004250212,0.001020484,0.999338931,0.036091477],[-1,0,1,0],[9E+09,9E+09,9E+09,9E+09,9E+09,9E+09]];
  CONST robtarget pGluePath1_180:=[[628.728252839,1115.671688615,-28.725179075],[0.004257408,0.000987638,0.999030385,0.043808538],[-1,0,1,0],[9E+09,9E+09,9E+09,9E+09,9E+09,9E+09]];
  CONST robtarget pGluePath1_190:=[[600.63785036,1237.2981322,-16.626015616],[0.004269192,0.000930981,0.998360233,0.057076724],[-1,0,1,0],[9E+09,9E+09,9E+09,9E+09,9E+09,9E+09]];
  CONST robtarget pGluePath1_200:=[[588.829791018,1275.073408124,-12.228310095],[0.004272683,0.000913448,0.998117695,0.061171701],[-1,0,1,0],[9E+09,9E+09,9E+09,9E+09,9E+09,9E+09]];
  CONST robtarget pGluePath1_210:=[[572.922506617,1307.138455712,-8.297892066],[0.004275529,0.000898824,0.99790276,0.064583227],[-1,0,1,0],[9E+09,9E+09,9E+09,9E+09,9E+09,9E+09]];
  CONST robtarget pGluePath1_220:=[[555.646456042,1323.034280615,-6.347032518],[0.004276856,0.000891926,0.997797398,0.066191126],[-1,0,1,0],[9E+09,9E+09,9E+09,9E+09,9E+09,9E+09]];
  CONST robtarget pGluePath1_230:=[[533.217965977,1329.408471018,-5.68440071],[0.004277385,0.000889163,0.997754477,0.066835005],[-1,0,1,0],[9E+09,9E+09,9E+09,9E+09,9E+09,9E+09]];
  CONST robtarget pGluePath1_240:=[[521.965807376,1330.190202116,-5.676774099],[0.004277187,0.0008888,0.997749085,0.06691546],[-1,0,1,0],[9E+09,9E+09,9E+09,9E+09,9E+09,9E+09]];
  CONST robtarget pGluePath1_250:=[[510.873367794,1330.321457852,-5.755848625],[0.004277462,0.000888769,0.997748318,0.066926884],[-1,0,1,0],[9E+09,9E+09,9E+09,9E+09,9E+09,9E+09]];
  CONST robtarget pGluePath2_10:=[[619.828545606,285.528137759,-43.361055016],[0.017445471,0.000804474,0.999029342,-0.040439867],[0,0,-2,0],[9E+09,9E+09,9E+09,9E+09,9E+09,9E+09]];
  CONST robtarget pGluePath2_20:=[[542.919099689,203.339057755,-38.406815989],[0.014160809,0.000898394,0.998793692,-0.047008782],[0,0,-2,0],[9E+09,9E+09,9E+09,9E+09,9E+09,9E+09]];
  CONST robtarget pGluePath2_30:=[[465.366451584,281.810603847,-47.283003108],[0.011025435,0.001063409,0.999107488,-0.040761959],[0,0,-2,0],[9E+09,9E+09,9E+09,9E+09,9E+09,9E+09]];
  CONST robtarget pGluePath3_10:=[[818.587593009,-12.950846089,-2.777508925],[0.025681178,0.00003066,0.997521056,-0.065515024],[0,0,-2,0],[9E+09,9E+09,9E+09,9E+09,9E+09,9E+09]];
  CONST robtarget pGluePath3_20:=[[818.737862458,80.629346079,-14.372847875],[0.025721235,0.000167153,0.998005837,-0.0576432],[0,0,-2,0],[9E+09,9E+09,9E+09,9E+09,9E+09,9E+09]];
  CONST robtarget pGluePath3_30:=[[818.921283452,174.37514383,-24.487731495],[0.025754438,0.000304173,0.998428619,-0.049768559],[0,0,-2,0],[9E+09,9E+09,9E+09,9E+09,9E+09,9E+09]];
  CONST robtarget pGluePath3_40:=[[819.137830741,268.268985324,-33.120448735],[0.025780733,0.000441599,0.998789415,-0.041891089],[0,0,-2,0],[9E+09,9E+09,9E+09,9E+09,9E+09,9E+09]];
  CONST robtarget pGluePath3_50:=[[819.387479075,362.293308742,-40.269288468],[0.02580006,0.000579306,0.999088229,-0.034010771],[0,0,-3,0],[9E+09,9E+09,9E+09,9E+09,9E+09,9E+09]];
  CONST robtarget pGluePath3_70:=[[819.495985813,441.995660701,-44.125910281],[0.010976994,-0.00136284,-0.999890974,0.009782089],[-1,0,-3,0],[9E+09,9E+09,9E+09,9E+09,9E+09,9E+09]];
  CONST robtarget pGluePath3_80:=[[814.684611714,516.212678859,-44.452584562],[0.011083874,-0.001794313,-0.999427173,0.03192576],[-1,0,-3,0],[9E+09,9E+09,9E+09,9E+09,9E+09,9E+09]];
  CONST robtarget pGluePath3_90:=[[816.795983092,553.341247437,-49.539467372],[0.024557104,0.000943952,0.999597469,-0.014175933],[-1,0,-3,0],[9E+09,9E+09,9E+09,9E+09,9E+09,9E+09]];
  CONST robtarget pGluePath3_100:=[[813.859673481,590.437316222,-50.605189936],[0.023534121,0.001013789,0.999667089,-0.010527495],[-1,0,-3,0],[9E+09,9E+09,9E+09,9E+09,9E+09,9E+09]];
  CONST robtarget pGluePath3_110:=[[811.286281422,614.062705666,-51.174312449],[0.022688853,0.001055035,0.999707841,-0.008266517],[-1,0,-3,0],[9E+09,9E+09,9E+09,9E+09,9E+09,9E+09]];
  CONST robtarget pGluePath3_120:=[[808.033625186,638.3744151,-51.672010261],[0.021699552,0.001093474,0.99974598,-0.005992385],[-1,0,-3,0],[9E+09,9E+09,9E+09,9E+09,9E+09,9E+09]];
  CONST robtarget pGluePath3_130:=[[804.226066637,662.263198877,-52.074391855],[0.020609841,0.001126548,0.999779671,-0.003817816],[-1,0,-3,0],[9E+09,9E+09,9E+09,9E+09,9E+09,9E+09]];
  CONST robtarget pGluePath3_140:=[[800.103144852,684.636024774,-52.373115157],[0.019493627,0.00115274,0.999807626,-0.001838892],[-1,0,-3,0],[9E+09,9E+09,9E+09,9E+09,9E+09,9E+09]];
  CONST robtarget pGluePath3_150:=[[796.006786893,704.422536026,-52.573859076],[0.018438738,0.001171739,0.999829296,-0.000136248],[-1,0,-3,0],[9E+09,9E+09,9E+09,9E+09,9E+09,9E+09]];
  CONST robtarget pGluePath3_160:=[[787.255006831,742.049116603,-52.774062397],[0.016902517,0.001200935,0.99985103,0.003283442],[-1,0,-3,0],[9E+09,9E+09,9E+09,9E+09,9E+09,9E+09]];
  CONST robtarget pGluePath3_170:=[[777.279910495,783.954371482,-52.65199767],[0.01609676,0.001230682,0.999841463,0.007511897],[-1,0,-3,0],[9E+09,9E+09,9E+09,9E+09,9E+09,9E+09]];
  CONST robtarget pGluePath3_180:=[[746.096040801,917.397780378,-49.791936443],[0.013084994,0.001269314,0.999697888,0.020767849],[-1,0,-3,0],[9E+09,9E+09,9E+09,9E+09,9E+09,9E+09]];
  CONST robtarget pGluePath3_190:=[[715.092241263,1050.67750445,-43.202958433],[0.010114919,0.001229016,0.999368538,0.03403974],[-1,0,-3,0],[9E+09,9E+09,9E+09,9E+09,9E+09,9E+09]];
  CONST robtarget pGluePath3_200:=[[684.299029926,1183.661977692,-32.893935771],[0.007193427,0.001111595,0.998853184,0.047321619],[-1,0,-3,0],[9E+09,9E+09,9E+09,9E+09,9E+09,9E+09]];
  CONST robtarget pGluePath3_210:=[[676.374413874,1217.111598476,-29.728806812],[0.005306942,0.001012871,0.998725127,0.050188948],[-1,0,-3,0],[9E+09,9E+09,9E+09,9E+09,9E+09,9E+09]];
  CONST robtarget pGluePath3_220:=[[670.344655396,1240.801609513,-27.365536588],[0.003271169,0.000901578,0.998647426,0.051882607],[-1,0,-3,0],[9E+09,9E+09,9E+09,9E+09,9E+09,9E+09]];
  CONST robtarget pGluePath3_230:=[[663.651139256,1264.844347399,-24.873922668],[0.00036384,0.000740454,0.998588416,0.053108334],[-1,0,-3,0],[9E+09,9E+09,9E+09,9E+09,9E+09,9E+09]];
  CONST robtarget pGluePath3_240:=[[656.343779136,1288.033792416,-22.396518605],[0.003669548,-0.000522469,-0.998566686,-0.053393218],[-1,0,-3,0],[9E+09,9E+09,9E+09,9E+09,9E+09,9E+09]];
  CONST robtarget pGluePath3_250:=[[652.298387039,1299.442241027,-21.158020729],[0.006289749,-0.000388958,-0.998577144,-0.052952569],[-1,0,-3,0],[9E+09,9E+09,9E+09,9E+09,9E+09,9E+09]];
  CONST robtarget pGluePath3_260:=[[647.912178867,1310.672870044,-19.931773606],[0.009413019,-0.000242469,-0.99860822,-0.051893731],[-1,0,-3,0],[9E+09,9E+09,9E+09,9E+09,9E+09,9E+09]];
  CONST robtarget pGluePath3_270:=[[643.38988111,1321.054998276,-18.797440616],[0.012879727,-0.000101479,-0.998662396,-0.050075154],[-1,0,-3,0],[9E+09,9E+09,9E+09,9E+09,9E+09,9E+09]];
  CONST robtarget pGluePath3_280:=[[639.007689653,1330.018887453,-17.823187036],[0.016380669,0.000010062,-0.99873604,-0.047518382],[-1,0,-3,0],[9E+09,9E+09,9E+09,9E+09,9E+09,9E+09]];
  CONST robtarget pGluePath3_290:=[[634.73508751,1337.789727295,-16.987973088],[0.019798791,0.000078268,-0.998826544,-0.044198826],[-1,0,-3,0],[9E+09,9E+09,9E+09,9E+09,9E+09,9E+09]];
  CONST robtarget pGluePath3_300:=[[630.516582844,1344.595264391,-16.268980735],[0.023017475,0.00009019,-0.998931493,-0.040075677],[-1,0,-3,0],[9E+09,9E+09,9E+09,9E+09,9E+09,9E+09]];
  CONST robtarget pGluePath3_310:=[[623.850400985,1353.755657883,-15.335116208],[0.027455683,-0.0000445,-0.9991296,-0.031404232],[-1,0,-3,0],[9E+09,9E+09,9E+09,9E+09,9E+09,9E+09]];
  CONST robtarget pGluePath3_320:=[[618.005243708,1360.267301456,-14.711773853],[0.02984968,-0.000331894,-0.999312992,-0.021964312],[-1,0,-3,0],[9E+09,9E+09,9E+09,9E+09,9E+09,9E+09]];
  CONST robtarget pGluePath3_330:=[[614.353373777,1363.740587594,-14.394533426],[0.03033333,-0.000547026,-0.999409136,-0.016154546],[-1,0,-3,0],[9E+09,9E+09,9E+09,9E+09,9E+09,9E+09]];
  CONST robtarget pGluePath3_340:=[[610.046597921,1367.353839634,-14.078595643],[0.030027464,-0.00080445,-0.999502649,-0.00959997],[-1,0,-3,0],[9E+09,9E+09,9E+09,9E+09,9E+09,9E+09]];
  CONST robtarget pGluePath3_350:=[[604.950784528,1371.058567861,-13.773104],[0.028653177,-0.001082859,-0.999585817,-0.002452959],[-1,0,-3,0],[9E+09,9E+09,9E+09,9E+09,9E+09,9E+09]];
  CONST robtarget pGluePath3_360:=[[598.934451197,1374.769964944,-13.49133823],[0.025989235,-0.001344248,-0.999649041,0.00495459],[-1,0,-3,0],[9E+09,9E+09,9E+09,9E+09,9E+09,9E+09]];
  CONST robtarget pGluePath3_370:=[[591.990047784,1378.322165384,-13.252944519],[0.022052352,-0.001540314,-0.999683139,0.012039255],[-1,0,-3,0],[9E+09,9E+09,9E+09,9E+09,9E+09,9E+09]];
  CONST robtarget pGluePath3_380:=[[584.106608273,1381.585030576,-13.073605251],[0.017107835,-0.001640087,-0.999684836,0.018299223],[-1,0,-3,0],[9E+09,9E+09,9E+09,9E+09,9E+09,9E+09]];
  CONST robtarget pGluePath3_390:=[[575.005055357,1384.538057527,-12.963300319],[0.011427017,-0.001639782,-0.999655984,0.023550957],[-1,0,-3,0],[9E+09,9E+09,9E+09,9E+09,9E+09,9E+09]];
  CONST robtarget pGluePath3_400:=[[564.437484441,1387.104459393,-12.937955988],[0.00541424,-0.001554309,-0.999601821,0.02764906],[-1,0,-3,0],[9E+09,9E+09,9E+09,9E+09,9E+09,9E+09]];
  CONST robtarget pGluePath3_410:=[[552.693648296,1389.11308473,-13.010127399],[0.000241056,0.001420698,0.999534148,-0.030486231],[-1,0,-3,0],[9E+09,9E+09,9E+09,9E+09,9E+09,9E+09]];
  CONST robtarget pGluePath3_420:=[[541.259586496,1390.409260874,-13.15804872],[0.004689967,0.001290956,0.999471379,-0.032144989],[-1,0,-3,0],[9E+09,9E+09,9E+09,9E+09,9E+09,9E+09]];
  CONST robtarget pGluePath3_430:=[[530.307719723,1391.175024699,-13.354520903],[0.008078771,0.001182158,0.999418499,-0.033105896],[-1,0,-3,0],[9E+09,9E+09,9E+09,9E+09,9E+09,9E+09]];
  CONST robtarget pGluePath3_440:=[[519.884010249,1391.560578756,-13.579672335],[0.010630504,0.001096314,0.999375942,-0.033667733],[-1,0,-3,0],[9E+09,9E+09,9E+09,9E+09,9E+09,9E+09]];
  CONST robtarget pGluePath3_450:=[[325.010254489,1391.98806787,-17.009312501],[0.00464115,0.001299272,0.999410474,-0.033992303],[-1,0,-3,0],[9E+09,9E+09,9E+09,9E+09,9E+09,9E+09]];
  CONST robtarget pGluePath3_460:=[[139.957935384,1392.495674153,-17.282760925],[0.003254996,-0.001567803,-0.999415921,0.033981826],[-1,0,-3,0],[9E+09,9E+09,9E+09,9E+09,9E+09,9E+09]];
  CONST robtarget pGluePath3_470:=[[-45.068908715,1393.199973641,-14.638993765],[0.011150468,-0.001836236,-0.999358983,0.033969388],[-1,0,-3,0],[9E+09,9E+09,9E+09,9E+09,9E+09,9E+09]];
  CONST robtarget pGluePath3_480:=[[-156.141315138,1393.679848356,-12.205656428],[0.01101736,-0.001831711,-0.999360459,0.033969616],[-1,0,-3,0],[9E+09,9E+09,9E+09,9E+09,9E+09,9E+09]];
  CONST robtarget pGluePath3_490:=[[-161.118318722,1392.724613331,-12.284659134],[0.031208357,0.000445256,0.999005758,-0.031832922],[-1,0,-3,0],[9E+09,9E+09,9E+09,9E+09,9E+09,9E+09]];
  CONST robtarget pGluePath3_500:=[[-165.364544134,1389.960189403,-12.509424244],[0.059972892,0.001127024,0.998198945,-0.000921483],[-1,0,-3,0],[9E+09,9E+09,9E+09,9E+09,9E+09,9E+09]];
  CONST robtarget pGluePath3_510:=[[-168.252754392,1385.783392839,-12.842509854],[0.058493568,0.003250874,0.997422849,0.041419742],[-1,-1,-3,0],[9E+09,9E+09,9E+09,9E+09,9E+09,9E+09]];
  CONST robtarget pGluePath3_520:=[[-169.311363369,1380.796428721,-13.229635335],[0.026966475,0.002472692,0.99716194,0.070247847],[-1,-1,-3,0],[9E+09,9E+09,9E+09,9E+09,9E+09,9E+09]];
  CONST robtarget pGluePath3_530:=[[-169.439588264,1363.446405379,-15.660797665],[0.026969813,0.002439673,0.997286871,0.068451249],[-1,-1,-3,0],[9E+09,9E+09,9E+09,9E+09,9E+09,9E+09]];
  CONST robtarget pGluePath3_550:=[[-169.975777315,1272.297603849,-23.387187829],[0.026810494,0.002284905,0.997798845,0.060608924],[-1,-1,-3,0],[9E+09,9E+09,9E+09,9E+09,9E+09,9E+09]];
  CONST robtarget pGluePath3_560:=[[-170.448587366,1203.094724156,-31.316397613],[0.026668126,0.002138868,0.998233164,0.053054564],[-1,-1,-3,0],[9E+09,9E+09,9E+09,9E+09,9E+09,9E+09]];
  CONST robtarget pGluePath3_570:=[[-170.89882643,1133.779418305,-38.195743096],[0.026536712,0.001995512,0.998609864,0.04549901],[-1,-1,-3,0],[9E+09,9E+09,9E+09,9E+09,9E+09,9E+09]];
  CONST robtarget pGluePath3_580:=[[-171.32642092,1064.367704912,-44.023797405],[0.026416141,0.001854524,0.998929043,0.037940952],[-1,-1,-3,0],[9E+09,9E+09,9E+09,9E+09,9E+09,9E+09]];
  CONST robtarget pGluePath3_590:=[[-171.731293901,994.875581484,-48.799180731],[0.026306321,0.001715613,0.999190712,0.030380194],[-1,-1,-3,0],[9E+09,9E+09,9E+09,9E+09,9E+09,9E+09]];
  CONST robtarget pGluePath3_600:=[[-172.113356646,925.318966676,-52.520774558],[0.026207183,0.001578506,0.999394853,0.022817101],[-1,-1,-3,0],[9E+09,9E+09,9E+09,9E+09,9E+09,9E+09]];
  CONST robtarget pGluePath3_610:=[[-172.472517865,855.713760444,-55.187543943],[0.026118659,0.0014429,0.999541474,0.015250407],[-1,0,-3,0],[9E+09,9E+09,9E+09,9E+09,9E+09,9E+09]];
  CONST robtarget pGluePath3_620:=[[-172.808686254,786.075862778,-56.798453969],[0.0260407,0.001308497,0.999630534,0.007678849],[-1,0,-3,0],[9E+09,9E+09,9E+09,9E+09,9E+09,9E+09]];
  CONST robtarget pGluePath3_630:=[[-173.283365614,707.221567257,-61.794666554],[0.026343708,0.001736188,0.999156009,0.031468452],[-1,-1,-3,0],[9E+09,9E+09,9E+09,9E+09,9E+09,9E+09]];
  CONST robtarget pGluePath3_640:=[[-173.645702816,621.481268031,-61.29631298],[0.025917312,0.001044583,0.999636574,-0.007343156],[-1,0,-3,0],[9E+09,9E+09,9E+09,9E+09,9E+09,9E+09]];
  CONST robtarget pGluePath3_650:=[[-173.972297328,535.761986461,-59.29812891],[0.025864563,0.000892019,0.999535666,-0.016083556],[-1,0,-3,0],[9E+09,9E+09,9E+09,9E+09,9E+09,9E+09]];
  CONST robtarget pGluePath3_660:=[[-174.265882207,450.064261991,-55.797984466],[0.025825778,0.00073964,0.999357881,-0.024825546],[-1,0,-3,0],[9E+09,9E+09,9E+09,9E+09,9E+09,9E+09]];
  CONST robtarget pGluePath3_670:=[[-174.526355204,364.406926002,-50.794929052],[0.02580006,0.000579308,0.999088233,-0.034010658],[0,0,-2,0],[9E+09,9E+09,9E+09,9E+09,9E+09,9E+09]];
  CONST robtarget pGluePath3_680:=[[-174.776003306,270.365273959,-43.644580035],[0.025780781,0.000441578,0.998789369,-0.041892164],[0,0,-2,0],[9E+09,9E+09,9E+09,9E+09,9E+09,9E+09]];
  CONST robtarget pGluePath3_690:=[[-174.992571432,176.452164045,-35.009604925],[0.025754634,0.000304136,0.998428536,-0.049770126],[0,0,-2,0],[9E+09,9E+09,9E+09,9E+09,9E+09,9E+09]];
  CONST robtarget pGluePath3_700:=[[-175.176017703,82.687166625,-24.89195247],[0.02572167,0.000167095,0.998005718,-0.057645068],[0,0,-2,0],[9E+09,9E+09,9E+09,9E+09,9E+09,9E+09]];
  CONST robtarget pGluePath3_710:=[[-175.326300239,-10.910147998,-13.293571511],[0.025681946,0.000030566,0.997520874,-0.065517502],[0,0,-2,0],[9E+09,9E+09,9E+09,9E+09,9E+09,9E+09]];
  CONST robtarget pGluePath3_720:=[[-174.342539685,-15.875836632,-12.637272121],[0.020454415,0.000530707,0.998394111,-0.052825505],[0,0,-2,0],[9E+09,9E+09,9E+09,9E+09,9E+09,9E+09]];
  CONST robtarget pGluePath3_730:=[[-171.510214446,-20.096144227,-12.077611404],[0.007638405,0.0012056,0.998843936,-0.047444632],[0,0,-2,0],[9E+09,9E+09,9E+09,9E+09,9E+09,9E+09]];
  CONST robtarget pGluePath3_740:=[[-167.264026403,-22.925098659,-11.700973139],[0.005397553,-0.001896241,-0.998595863,0.052664721],[0,0,-2,0],[9E+09,9E+09,9E+09,9E+09,9E+09,9E+09]];
  CONST robtarget pGluePath3_750:=[[-162.252702234,-23.919359122,-11.567891538],[0.011003597,-0.002440215,-0.997786342,0.065539157],[0,0,-2,0],[9E+09,9E+09,9E+09,9E+09,9E+09,9E+09]];
  CONST robtarget pGluePath3_760:=[[-51.178860591,-24.399231504,-14.001162731],[0.011003549,-0.002440293,-0.997786067,0.065543355],[0,0,-2,0],[9E+09,9E+09,9E+09,9E+09,9E+09,9E+09]];
  CONST robtarget pGluePath3_770:=[[163.029446779,-25.196914614,-16.795832158],[0.002028744,-0.001850168,-0.997847959,0.065512688],[0,0,-2,0],[9E+09,9E+09,9E+09,9E+09,9E+09,9E+09]];
  CONST robtarget pGluePath3_780:=[[377.235422177,-25.730710016,-15.680759907],[0.007078893,0.001252113,0.997826848,-0.065497355],[0,0,-2,0],[9E+09,9E+09,9E+09,9E+09,9E+09,9E+09]];
  CONST robtarget pGluePath3_790:=[[591.385387932,-26.000373579,-10.656718624],[0.016186046,0.000654315,0.997721215,-0.0654978],[0,0,-2,0],[9E+09,9E+09,9E+09,9E+09,9E+09,9E+09]];
  CONST robtarget pGluePath3_800:=[[805.425602441,-26.005661494,-1.724484244],[0.025292626,0.000056197,0.997531051,-0.065513983],[0,0,-2,0],[9E+09,9E+09,9E+09,9E+09,9E+09,9E+09]];
  CONST robtarget pGluePath3_810:=[[810.449420554,-25.012122362,-1.598951077],[0.025225832,0.000057342,0.997520354,-0.065702345],[0,0,-2,0],[9E+09,9E+09,9E+09,9E+09,9E+09,9E+09]];
  CONST robtarget pGluePath3_820:=[[814.721031137,-22.175159511,-1.756004459],[0.025353078,0.000046534,0.997507899,-0.065842311],[0,0,-2,0],[9E+09,9E+09,9E+09,9E+09,9E+09,9E+09]];
  CONST robtarget pGluePath3_830:=[[817.582604011,-17.937177715,-2.170191722],[0.025573333,0.000033176,0.997506711,-0.065775115],[0,0,-2,0],[9E+09,9E+09,9E+09,9E+09,9E+09,9E+09]];
  CONST robtarget pGluePath3_840:=[[818.587592225,-12.951369525,-2.77743986],[0.025681179,0.00003066,0.997521056,-0.065515024],[0,0,-2,0],[9E+09,9E+09,9E+09,9E+09,9E+09,9E+09]];
  CONST robtarget pGluePath3_850:=[[818.737862458,80.629346079,-14.372847875],[0.025721235,0.000167153,0.998005837,-0.0576432],[0,0,-2,0],[9E+09,9E+09,9E+09,9E+09,9E+09,9E+09]];
  CONST robtarget pGluePath3_860:=[[818.921283452,174.37514383,-24.487731495],[0.025754438,0.000304173,0.998428619,-0.049768559],[0,0,-2,0],[9E+09,9E+09,9E+09,9E+09,9E+09,9E+09]];
  CONST robtarget pGluePath3_870:=[[819.137830741,268.268985324,-33.120448735],[0.025780733,0.000441599,0.998789415,-0.041891089],[0,0,-2,0],[9E+09,9E+09,9E+09,9E+09,9E+09,9E+09]];
  CONST robtarget pGluePath3_880:=[[819.387479075,362.293308742,-40.269288468],[0.02580006,0.000579306,0.999088229,-0.034010771],[0,0,-3,0],[9E+09,9E+09,9E+09,9E+09,9E+09,9E+09]];
  CONST robtarget pApproach_Path1:=[[510.024254477,1316.966975761,93.344792556],[0.004277461,0.000888769,0.997748318,0.066926884],[-1,0,1,0],[9E+09,9E+09,9E+09,9E+09,9E+09,9E+09]];
  CONST robtarget pApproach_Path2:=[[619.828545606,285.528137759,-43.361055016],[0.017445471,0.000804474,0.999029342,-0.040439867],[0,0,-2,0],[9E+09,9E+09,9E+09,9E+09,9E+09,9E+09]];
  CONST robtarget pDepart_Path2:=[[465.366451584,281.810603847,-47.283003108],[0.011025435,0.001063409,0.999107488,-0.040761959],[0,0,-2,0],[9E+09,9E+09,9E+09,9E+09,9E+09,9E+09]];
  CONST robtarget pApproach_Path3:=[[818.587593009,-12.950846089,-2.777508925],[0.025681178,0.00003066,0.997521056,-0.065515024],[0,0,-2,0],[9E+09,9E+09,9E+09,9E+09,9E+09,9E+09]];
  CONST robtarget pDepart_Path3:=[[819.387479075,362.293308742,-40.269288468],[0.02580006,0.000579306,0.999088229,-0.034010771],[0,0,-3,0],[9E+09,9E+09,9E+09,9E+09,9E+09,9E+09]];
  CONST robtarget pDepart_Path1:=[[510.007905183,1316.966981005,93.344650479],[0.004277462,0.000888769,0.997748318,0.066926884],[-1,0,1,0],[9E+09,9E+09,9E+09,9E+09,9E+09,9E+09]];
ENDMODULE

! task T_ROB1
MODULE modCalibData
  PERS tooldata tNozzle:=[TRUE,[[-305.801192078,0,351.776515421],[0.991444861,0,-0.130526192,0]],[10,[-216.957886762,-4.684934403,103.554004337],[1,0,0,0],0,0,0]];
  TASK PERS wobjdata wobjDockingStn:=[FALSE,TRUE,"",[[93.58826629,-1285.222736121,827.125],[0.818981032,0,0,-0.57382059]],[[0,0,0],[1,0,0,0]]];
ENDMODULE

! task T_ROB1
MODULE modRobotStudio
  CONST robtarget pDockingStn:=[[-6.21722435,13.985562095,-127.5],[0,0.737075919,0.675809951,0],[-1,0,0,0],[9E+09,9E+09,9E+09,9E+09,9E+09,9E+09]];
  CONST robtarget pAboveDockingStn:=[[-6.217297914,13.985583992,22.500016978],[-0.000000026,0.737075879,0.675809995,-0.000000022],[-1,0,0,0],[9E+09,9E+09,9E+09,9E+09,9E+09,9E+09]];
  PROC FromDockingStation()
    MoveJ pDockingStn,v200,z1,tNozzle\WObj:=wobjDockingStn;
    MoveL pAboveDockingStn,v200,z1,tNozzle\WObj:=wobjDockingStn;
  ENDPROC
  PROC ToDockingStation()
    MoveL pAboveDockingStn,v1000,z1,tNozzle\WObj:=wobjDockingStn;
    MoveL pDockingStn,v200,fine,tNozzle\WObj:=wobjDockingStn;
  ENDPROC
ENDMODULE

